Fanuc KAREL source: kc00035.KL

-- PROVISIONAL review KL for V1013-1; original PC SHA256 f88a0575c068f710adc22d980f08b5cf115f86a06bfea73a1014a35c6c8c3e1d
-- Incomplete behavior may be omitted. Consult companion uncertainty JSON. Do not deploy.
PROGRAM KC00035
%NOLOCKGROUP
BEGIN
  -- UNRESOLVED_PC offsets 5-41; opcodes 27,22,22,2A,22,22,22,31
  -- UNRESOLVED_PC offsets 46-50; opcodes 7F
END KC00035
